// TwinCAT 3 PLC project Gesamtsystemebene
// ProgramVersion: 3.1.4024.0
// libraries:
//   Tc2_Standard, * (Beckhoff Automation GmbH)
//   Tc2_System, * (Beckhoff Automation GmbH)
//   Tc3_Module, * (Beckhoff Automation GmbH)
//   Tc3_PLCopen_OpcUa, * (Beckhoff Automation GmbH)
//   VisuDialogs, * (System)
//   Tc2_OpcUa,3.3.2.0,Beckhoff Automation GmbH
// project tree:
//   DUTs/01_Schnittstellen/ I_Auswertung.TcIO, I_Reaktor.TcIO
//   DUTs/02_Strukturen/ LeitungControlWord.TcDUT, RezeptControlWord.TcDUT, RezeptStatusWord.TcDUT (not stored), SekControlWord.TcDUT (not stored), SystemStatusWord.TcDUT
//   / GlobalTextList.TcGTLO, PlcTask.TcTTO, Visualisierungsmanager.TcVMO (not stored), VISU_TASK.TcTTO
//   GVLs/01_OPC_UA/ GVL_OPC_UA.TcGVL
//   GVLs/ GVL.TcGVL
//   POUs/01_Rezept/ Rezept_1.TcPOU
//   POUs/02_Funktionsblock/ FB_Auswertung.TcPOU, FB_Reaktoreinheit.TcPOU, FB_UpdateHandler.TcPOU
//   POUs/03_System/ Reaktoranlage.TcPOU, Systemauswertung.TcPOU
//   POUs/04_Abläufe/01_Vererbung/ FB_Basis.TcPOU
//   POUs/04_Abläufe/ FB_Lesen.TcPOU, FB_Trennen.TcPOU, FB_UpdateSek.TcPOU, FB_UpdateSys.TcPOU, FB_Verbinden.TcPOU, FB_Grundablauf.TcPOU
//   POUs/05_Kommunikation/ Connect.TcPOU, Disconnect.TcPOU, Read.TcPOU, UpdateSek.TcPOU, UpdateSys.TcPOU
//   POUs/ MAIN.TcPOU
//   VISUs/ Test_Visu.TcVIS
// real-time tasks:
//   TASK PlcTask: cycle T#10ms, priority 20, ADS port 350
//   TASK VISU_TASK: cycle T#200000us, priority 30, ADS port 351
//   TASK Gerät 1 (OPC UA Virtual)_Task_58: cycle T#40ms, priority 58, ADS port 352

CONFIGURATION Gesamtsystemebene
    RESOURCE PLC ON TwinCAT3
        TASK PlcTask(INTERVAL := T#10ms, PRIORITY := 20);
        TASK VISU_TASK(INTERVAL := T#200000us, PRIORITY := 30);
        PROGRAM MAIN WITH PlcTask : MAIN;
        PROGRAM VisuElems_Visu_Prg WITH VISU_TASK : VisuElems.Visu_Prg;
    END_RESOURCE
END_CONFIGURATION

// ---- DUTs/02_Strukturen/LeitungControlWord.TcDUT
TYPE LeitungControlWord :
STRUCT
	A_Prueft			:BOOL;
	A_Besetzt			:BOOL;
	B_Prueft			:BOOL;
	B_Besetzt			:BOOL;
	C_Prueft			:BOOL;
	C_Besetzt			:BOOL;
	D_Prueft			:BOOL;
	D_Besetzt			:BOOL;
	E_Prueft			:BOOL;
	E_Besetzt			:BOOL;
	F_Prueft			:BOOL;
	F_Besetzt			:BOOL;
END_STRUCT
END_TYPE

// ---- DUTs/02_Strukturen/RezeptControlWord.TcDUT
TYPE RezeptControlWord :
STRUCT			
	PowerOn			:BOOL;			// Einschalten von Reaktoreinheit
	SekReakt		:INT;			// Definierter sekundär-Reaktor
	Leitung			:INT;			// Definiert welche Leitung verwendet wird
	Temp			:REAL;			// Definierte Temperatur für Heiz- / Kühlprozess
	Enlteermenge	:REAL;			// Zu entleerende Menge
	Pumpmenge		:REAL;			// Zu pumpende Menge
	Haltedauer		:INT;			// Wie lange soll Temperatur gehalten werden (Faktor für Sekunden)
	Ruehrdauer		:INT;			// Wie lange soll gerührt werden (Faktor für Sekunden)
	Wartedauer		:INT;			// Wie lange soll gerührt werden (Faktor für Sekunden)
	Zirkulierdauer	:INT;			// Wie lange soll zirkuliert werden (Faktor für Sekunden)
END_STRUCT
END_TYPE

// ---- DUTs/02_Strukturen/SystemStatusWord.TcDUT
TYPE SystemStatusWord :
STRUCT
	// Das SystemStatusWord ist für die Interaktion zwischen den Reaktoren 	

	// Reaktor 1
	R1_Ready		:BOOL;
	R1_Activ		:BOOL;
	// Reaktor 2
	R2_Ready		:BOOL;
	R2_Activ		:BOOL;
	// Reaktor 3
	R3_Ready		:BOOL;
	R3_Activ		:BOOL;
	// Reaktor 4
	R4_Ready		:BOOL;
	R4_Activ		:BOOL;
	// Reaktor 5
	R5_Ready		:BOOL;
	R5_Activ		:BOOL;
	// Reaktor 6
	R6_Ready		:BOOL;
	R6_Activ		:BOOL;
	// Reaktor 7
	R7_Ready		:BOOL;
	R7_Activ		:BOOL;
END_STRUCT	
END_TYPE

// ---- GVLs/01_OPC_UA/GVL_OPC_UA.TcGVL
{attribute 'qualified_only'}
VAR_GLOBAL
	// Verbindungsinformationen
	IP 				:ARRAY [0..6] OF STRING := [
		        'opc.tcp://169.254.240.1:4840', 
        		'opc.tcp://169.254.240.2:4840',
				'opc.tcp://169.254.240.3:4840', 
				'opc.tcp://169.254.240.4:4840', 
				'opc.tcp://169.254.240.5:4840', 
 				'opc.tcp://169.254.240.6:4840', 
        		'opc.tcp://169.254.240.7:4840'];	
	NameSpace		:STRING(MAX_STRING_LENGTH) := 'urn:BeckhoffAutomation:Ua:PLC1';
	ConnectionHdl	:ARRAY [0..6] OF DWORD := [];
END_VAR

// ---- GVLs/GVL.TcGVL
{attribute 'qualified_only'}
VAR_GLOBAL
		
	// Rezeptparameter
	R1_CW			:RezeptControlWord;				// Lokale definierung der Parameter
	R1_SW			:RezeptStatusWord;				// Statusword für internen Handling
	
	R2_CW			:RezeptControlWord;				// Lokale definierung der Parameter
	R2_SW			:RezeptStatusWord;				// Statusword für internen Handling
	
	R3_CW			:RezeptControlWord;				// Lokale definierung der Parameter
	R3_SW			:RezeptStatusWord;				// Statusword für internen Handling
	
	R4_CW			:RezeptControlWord;				// Lokale definierung der Parameter
	R4_SW			:RezeptStatusWord;				// Statusword für internen Handling
	
	R5_CW			:RezeptControlWord;				// Lokale definierung der Parameter
	R5_SW			:RezeptStatusWord;				// Statusword für internen Handling
	
	R6_CW			:RezeptControlWord;				// Lokale definierung der Parameter
	R6_SW			:RezeptStatusWord;				// Statusword für internen Handling
	
	R7_CW			:RezeptControlWord;				// Lokale definierung der Parameter
	R7_SW			:RezeptStatusWord;				// Statusword für internen Handling
	
	
	// Leitungs-Control-Word
	
	// SekundärControlWord
	SekControlWord	:SekControlWord;

	// SystemStatusWord
	SysStatusWord	:SystemStatusWord;
	
	// Funktionsvariablen
	// 0 = System nicht verbunden
	// 1 = System teilweisen Verbunden (Nicht Aktiv)
	// 2 = System Aktiv (Prozess läuft)
	// 9 = Error
	SysState		:INT;						
	
	// Bedienparameter 
	Start			:BOOL;
	Connect			:BOOL;
	Disconnect		:BOOL;
	Read			:BOOL;
	
	SekUpdate_1		:BOOL;
	SekUpdate_2		:BOOL;
	SekUpdate_3		:BOOL;
	SekUpdate_4		:BOOL;
	SekUpdate_5		:BOOL;
	SekUpdate_6		:BOOL;
	SekUpdate_7		:BOOL;
	SysUpdate_1		:BOOL;
	SysUpdate_2		:BOOL;
	SysUpdate_3		:BOOL;
	SysUpdate_4		:BOOL;
	SysUpdate_5		:BOOL;
	SysUpdate_6		:BOOL;
	SysUpdate_7		:BOOL;
	SekUpdateReset	:BOOL;
	SysUpdateReset	:BOOL;
	
	
	// Zustands-Variablen
	Error			:BOOL;
	ErrorID			:DWORD;
	
END_VAR

// ---- DUTs/01_Schnittstellen/I_Auswertung.TcIO
INTERFACE I_Auswertung

METHOD M_STATUS_SEK : BOOL
VAR_INPUT
END_VAR
END_METHOD

METHOD M_STATUS_SYSTEM : BOOL
VAR_INPUT
END_VAR
END_METHOD

METHOD M_TRENNEN : BOOL
VAR_INPUT
END_VAR
END_METHOD

METHOD M_VERBINDEN : BOOL
VAR_INPUT
END_VAR
END_METHOD

PROPERTY P_Status : INT
GET
END_GET
END_PROPERTY

END_INTERFACE

// ---- DUTs/01_Schnittstellen/I_Reaktor.TcIO
INTERFACE I_Reaktor

METHOD M_LESEN : BOOL
VAR_INPUT
END_VAR
END_METHOD

METHOD M_SCHREIBEN : BOOL
VAR_INPUT
END_VAR
END_METHOD

METHOD M_TRENNEN : BOOL
VAR_INPUT
END_VAR
END_METHOD

METHOD M_VERBINDEN : BOOL
VAR_INPUT
END_VAR
END_METHOD

METHOD M_ZUSTAND : BOOL
VAR_INPUT
END_VAR
END_METHOD

PROPERTY P_Status : INT
GET
END_GET
END_PROPERTY

END_INTERFACE

// ---- POUs/MAIN.TcPOU
PROGRAM MAIN
VAR
END_VAR

VAR_INPUT
END_VAR

// Starten der Anlage
Reaktoranlage();
Systemauswertung();

// Starten des Kommunikationsauswertung
Connect();
Disconnect();

// Lesen von RezeptStatusWord
Read();

// Auswertung des RezeptControlWords für Sekundärreaktor
UpdateSek();

// Auswertung des RezeptStatusWords für Systemupdate
UpdateSys();

// Starten des Rezeptes
Rezept_1();

END_PROGRAM

// ---- POUs/03_System/Reaktoranlage.TcPOU
PROGRAM Reaktoranlage
VAR
	R1				:FB_Reaktoreinheit;
	R2				:FB_Reaktoreinheit;
	
	// Instanziierung von Switchfunktion für Update-Variable
	Switch_R1		:FB_UpdateHandler;
	Switch_R2		:FB_UpdateHandler;
	Switch_R3		:FB_UpdateHandler;
	Switch_R4		:FB_UpdateHandler;
	Switch_R5		:FB_UpdateHandler;
	Switch_R6		:FB_UpdateHandler;
	Switch_R7		:FB_UpdateHandler;
END_VAR

Switch_R1(
    I_SekUpdate := R1.O_SekUpdate,
    I_SekReset := GVL.SekUpdateReset,
    I_SysUpdate := R1.O_SysUpdate,
    I_SysReset := GVL.SysUpdateReset); // FB_UpdateHandler
GVL.ErrorID := R1.O_ErrorID;
GVL_OPC_UA.ConnectionHdl[0] := R1.O_ConnectionHdl;
GVL.SekUpdate_1 := Switch_R1.O_SekUpdate;
R2(I_RNr := 2, I_IP := GVL_OPC_UA.IP, I_NameSpace := GVL_OPC_UA.NameSpace, I_CW := GVL.R2_CW); // FB_Reaktoreinheit
GVL.Error := R2.O_Error;
GVL.ErrorID := R2.O_ErrorID;
GVL.R2_SW := R2.O_SW;
GVL_OPC_UA.ConnectionHdl[1] := R2.O_ConnectionHdl;
GVL.SekUpdate_2 := Switch_R2.O_SekUpdate;
Switch_R2(
    I_SekUpdate := R2.O_SekUpdate,
    I_SekReset := GVL.SekUpdateReset,
    I_SysUpdate := R2.O_SysUpdate,
    I_SysReset := GVL.SysUpdateReset); // FB_UpdateHandler
GVL.SysUpdate_1 := Switch_R1.O_SysUpdate;
GVL.SysUpdate_2 := Switch_R2.O_SysUpdate;
R1(I_RNr := 1, I_IP := GVL_OPC_UA.IP, I_NameSpace := GVL_OPC_UA.NameSpace, I_CW := GVL.R1_CW); // FB_Reaktoreinheit
GVL.Error := R1.O_Error;
GVL.R1_SW := R1.O_SW;

END_PROGRAM

// ---- POUs/02_Funktionsblock/FB_Reaktoreinheit.TcPOU
FUNCTION_BLOCK FB_Reaktoreinheit IMPLEMENTS I_Reaktor
VAR_INPUT
	I_RNr					:INT;						// Nummer für korrekte Zuweisung von SystemStatusWord
	I_IP					:ARRAY [0..6] OF STRING;
	I_NameSpace				:STRING(MAX_STRING_LENGTH);
	I_CW					:RezeptControlWord;			// Variable für Kommunikations-Schnittstelle (Write)					
END_VAR
	
VAR_OUTPUT
	O_Verbunden				:BOOL;
	O_SekUpdate				:BOOL;
	O_SysUpdate				:BOOL;
	O_ConnectionHdl			:DWORD;
	O_Error					:BOOL;
	O_ErrorID				:DWORD;
	O_SW					:RezeptStatusWord; 			// Statusword für Kontrolle des Rezeptes 
END_VAR

VAR
	V_Status				:INT;						// Interne Variable
	OPC_Status				:INT;						// Variable für Verbindugsprozess
	Counter					:INT := 0;
	
	// Instanziierung der Kommunikationsfunktionsblöcke
	Connect					:UA_Connect;
	NameSpaceInd			:UA_GetNamespaceIndex;
	Node					:UA_NodeGetHandle;
	NodeRelease				:UA_NodeReleaseHandle;
	Disconnect				:UA_Disconnect;
	Status					:UA_ConnectGetStatus;
	Read					:UA_Read;	
	Write					:UA_Write;
	
	// Instanziierung der relevanten Input-Variablen
	ConnectInfo				:ST_UASessionConnectInfo;			// Informationen für Verbindungsaufbau 
	NodeID_SW				:ST_UANodeID;
	NodeID_CW				:ST_UANodeID;
	NodeIdentifier_SW		:STRING(MAX_STRING_LENGTH) := 'GVL_OPC_UA.SW';
	NodeIdentifier_CW 		:ARRAY [0..9] OF STRING := [
        'GVL_OPC_UA.CW.PowerOn', 
        'GVL_OPC_UA.CW.SekReakt', 
        'GVL_OPC_UA.CW.Leitung', 
        'GVL_OPC_UA.CW.Temp', 
        'GVL_OPC_UA.CW.Enlteermenge', 
        'GVL_OPC_UA.CW.Pumpmenge', 
        'GVL_OPC_UA.CW.Haltedauer', 
        'GVL_OPC_UA.CW.Ruehrdauer', 
        'GVL_OPC_UA.CW.Wartedauer', 
        'GVL_OPC_UA.CW.Zirkulierdauer'];
	
	// Instanziierung der relevanten Output-Variablen
	NameSpaceIndex			:UINT;
	NodeHdl_SW				:DWORD;						// Nodehandler für Statusword
	NodeHdl_CW 				:ARRAY [0..9] OF DWORD := [];
	ConnectionStatus		:E_UAConnectionStatus;
	ServerState				:E_UAServerState;
	
	O_Sek: INT;
END_VAR

// Setzen der internen Variablen
V_Status := P_Status;

// OPC-UA-Schnittstelle:
CASE OPC_Status OF
0: // Idle
	O_SekUpdate := FALSE;
	O_SysUpdate := FALSE;
1:	// Connect
	// Definition der Verbindungsinformationen
	ConnectInfo.tSessionTimeout := T#1M;
	ConnectInfo.tConnectTimeout := T#1M;
	ConnectInfo.sApplicationName := '';
	ConnectInfo.eSecurityMode := eUASecurityMsgMode_Sign_Encrypt;				// 3 = Sign_Encrypted
	ConnectInfo.eSecurityPolicyUri := eUASecurityPolicy_Basic256Sha256;			// 4 = Basic256  
	ConnectInfo.eTransportProfileUri := eUATransportProfileUri_UATcp;			// 1 = UATcp
	ConnectInfo.stUserIdentTokenType.eUserIdentTokenType := eUAUITT_Username;	// 1 = Username
	ConnectInfo.stUserIdentTokenType.sTokenParam1 := 'Administrator';			// Username
	ConnectInfo.stUserIdentTokenType.sTokenParam2 := '1';						// PW

	// Verbinden zu OPC-UA-Schnittstelle
	Connect(Execute := TRUE, 
			ServerUrl := I_IP[I_RNr - 1], 
			SessionConnectInfo := ConnectInfo, 
			Timeout := T#5S, 
			ConnectionHdl => O_ConnectionHdl, 
			Error => O_Error, 
			ErrorID => O_ErrorID);
			
	IF NOT Connect.Busy THEN
		Connect(Execute := FALSE);
	END_IF
			
	IF Connect.Error THEN
		O_Verbunden := FALSE;
		OPC_Status := 0;
	END_IF
			
	IF Connect.Done THEN
		OPC_Status := 2;
	END_IF
			
//==================================================================================================
2:	// NameSpaceIndex
	NameSpaceInd(Execute := TRUE,
				ConnectionHdl := O_ConnectionHdl,
				NameSpaceUri := I_NameSpace,
				Timeout := T#5S,
				NameSpaceIndex => NameSpaceIndex, 
				Error => O_Error, 
				ErrorID => O_ErrorID);
				
	IF NOT NameSpaceInd.Busy THEN
		NameSpaceInd(Execute := FALSE);
	END_IF
				
	IF NameSpaceInd.Error THEN
		O_Verbunden := FALSE;
		OPC_Status := 0;
	END_IF
	
	IF NameSpaceInd.Done THEN
		OPC_Status := 3;
	END_IF

//==================================================================================================				
3: // Nodes
	// Definieren von relevanten Parameter
	// RezeptStatusword - SW
	NodeID_SW.eIdentifierType := eUAIdentifierType_String;
	NodeID_SW.nNamespaceIndex := NameSpaceIndex;
	NodeID_SW.sIdentifier := NodeIdentifier_SW;
	
	// Definieren von SW Node
	Node(Execute := TRUE,
			ConnectionHdl := O_ConnectionHdl,
			NodeID := NodeID_SW,
			Timeout := T#5S,
			NodeHdl => NodeHdl_SW, 
			Error => O_Error, 
			ErrorID => O_ErrorID);

	IF NOT Node.Busy THEN
		Node(Execute := FALSE);
	END_IF 		
	
	IF Node.Error THEN
		OPC_Status := 0;
	END_IF
	
	IF Node.Done THEN
		OPC_Status := 4;
	END_IF

//==================================================================================================		
4:	// RezeptControlword
	// Die Node-Identifier jeder Variable werden einzeln in ein Array geschrieben. 
	// Innerhalb des Cases gibt es  einen Counter der die Arrayposition managed
	// Dafür braucht es keine For-Schleife, da der instanziierte FB zyklisch ausgeführt wird
	
	NodeID_CW.eIdentifierType := eUAIdentifierType_String;
	NodeID_CW.nNamespaceIndex := NameSpaceIndex;
	NodeID_CW.sIdentifier := NodeIdentifier_CW[Counter];
	
	Node(Execute := TRUE,
			ConnectionHdl := O_ConnectionHdl,
			NodeID := NodeID_CW,
			Timeout := T#5S,
			NodeHdl => NodeHdl_CW[Counter], 
			Error => O_Error, 
			ErrorID => O_ErrorID);
			
	IF NOT Node.Busy THEN
		Node(Execute := FALSE);
	END_IF		
	
	IF Node.Error THEN
		OPC_Status := 0;
	END_IF
	
	IF Node.Done AND Counter < 9 THEN
		Counter := Counter + 1;
	END_IF
	
	IF Node.Done AND Counter > 8 THEN // Muss angepasst werden wegen case 5
		OPC_Status := 0; 
		Counter := 0;	
		O_Verbunden := TRUE;
	END_IF	

//==================================================================================================	
5: // Lesen von Variablen
	Read(Execute := TRUE,
		ConnectionHdl := O_ConnectionHdl,
		NodeHdl := NodeHdl_SW,
		pVariable := ADR(O_SW),
		cbData := SIZEOF(O_SW),
		Timeout := T#5S,
		Error => O_Error,
		ErrorID => O_ErrorID);
	
	IF NOT Read.Busy THEN
		Read(Execute := FALSE);
	END_IF	
		
	IF Read.Error THEN
		OPC_Status := 0;
	END_IF
	
	IF Read.Done THEN
		OPC_Status := 0;
		IF O_SW.ReactReady OR O_SW.ReactActiv THEN
			O_SysUpdate := TRUE;
		END_IF
	END_IF
	
//==================================================================================================	
6: // Schreiben von Variablen		
	// Jede Variable in der Struktur muss separat berschrieben werden. 
	// Ansonsten werden die Daten nicht korrekt übertragen.
	
	CASE Counter OF 
		0: 		Write.pVariable := ADR(I_CW.PowerOn);
				Write.cbData  := SIZEOF(I_CW.PowerOn);
		1: 		Write.pVariable := ADR(I_CW.SekReakt);
				Write.cbData  := SIZEOF(I_CW.SekReakt);
		2: 		Write.pVariable := ADR(I_CW.Leitung);
				Write.cbData  := SIZEOF(I_CW.Leitung);
		3: 		Write.pVariable := ADR(I_CW.Temp);
				Write.cbData  := SIZEOF(I_CW.Temp);
		4: 		Write.pVariable := ADR(I_CW.Enlteermenge);
				Write.cbData  := SIZEOF(I_CW.Enlteermenge);
		5: 		Write.pVariable := ADR(I_CW.Pumpmenge);
				Write.cbData  := SIZEOF(I_CW.Pumpmenge);
		6: 		Write.pVariable := ADR(I_CW.Haltedauer);
				Write.cbData  := SIZEOF(I_CW.Haltedauer);
		7: 		Write.pVariable := ADR(I_CW.Ruehrdauer);
				Write.cbData  := SIZEOF(I_CW.Ruehrdauer);
		8: 		Write.pVariable := ADR(I_CW.Wartedauer);
				Write.cbData  := SIZEOF(I_CW.Wartedauer);
		9: 		Write.pVariable := ADR(I_CW.Zirkulierdauer);
				Write.cbData  := SIZEOF(I_CW.Zirkulierdauer);
	END_CASE
	
	Write(Execute := TRUE,
		ConnectionHdl := O_ConnectionHdl,
		NodeHdl := NodeHdl_CW[Counter],
		Timeout := T#5S,
		Error => O_Error,
		ErrorID => O_ErrorID);
	
	IF NOT Write.Busy THEN
		Write(Execute := FALSE);
	END_IF	
		
	IF Write.Error THEN
		OPC_Status := 0;
	END_IF
	
	IF Write.Done AND Counter < 9 THEN
		Counter := Counter + 1;
	END_IF
	
	IF Write.Done AND Counter > 8 THEN
		Counter := 0;
		OPC_Status := 0;
		IF I_CW.SekReakt > 0 THEN
			O_SekUpdate := TRUE;
		END_IF
	END_IF

//==================================================================================================	
7: // Release Node - RezeptStatusword
	NodeRelease(Execute := TRUE,
				ConnectionHdl := O_ConnectionHdl,
				NodeHdl := NodeHdl_SW,
				Timeout := T#5S,
				Error => O_Error,
				ErrorID => O_ErrorID);
	
	IF NOT NodeRelease.Busy THEN
		NodeRelease(Execute := FALSE);
	END_IF
	
	IF NodeRelease.Error THEN
		OPC_Status := 0;
	END_IF

	IF NodeRelease.Done THEN
		OPC_Status := 8;
	END_IF			

//==================================================================================================
8:	// Release Node - RezeptControlword
	NodeRelease(Execute := TRUE,
				ConnectionHdl := O_ConnectionHdl,
				NodeHdl := NodeHdl_CW[Counter],
				Timeout := T#5S,
				Error => O_Error,
				ErrorID => O_ErrorID);
	
	IF NOT NodeRelease.Busy THEN
		NodeRelease(Execute := FALSE);
	END_IF	
	
	IF NodeRelease.Error THEN
		OPC_Status := 0;
	END_IF

	IF NodeRelease.Done AND Counter < 9 THEN
		Counter := Counter + 1;
	END_IF				
				
	IF NodeRelease.Done AND Counter > 8 THEN
		OPC_Status := 9;
	END_IF
	
//==================================================================================================
9: // Disconnect
	Disconnect(Execute := TRUE,
				ConnectionHdl := O_ConnectionHdl,
				Timeout := T#5S,
				Error => O_Error,
				ErrorID => O_ErrorID);
	
	IF NOT Disconnect.Busy THEN
		Disconnect(Execute := FALSE);
	END_IF	

	IF Disconnect.Error THEN
		OPC_Status := 0;
	END_IF		
				
	IF Disconnect.Done THEN
		O_Verbunden := FALSE;
		OPC_Status := 0;
	END_IF	

//==================================================================================================
10: // Verbingungsstatus
	Status(Execute := TRUE,
			ConnectionHdl := O_ConnectionHdl,
			GetServiceLevel := FALSE,
			Timeout := T#5S,
			Error => O_Error,
			ErrorID => O_ErrorID,
			ConnectionStatus => ConnectionStatus,
			ServerState => ServerState);
	
	IF Status.Error THEN
		OPC_Status := 0;
	END_IF		
		
	IF Status.Done THEN
		Status(Execute := FALSE);
		OPC_Status := 0;
	END_IF
	
END_CASE

METHOD M_LESEN : BOOL
VAR_INPUT
END_VAR
OPC_Status := 5;

IF Read.Done THEN
	M_LESEN := TRUE;
END_IF
END_METHOD

METHOD M_SCHREIBEN : BOOL
VAR_INPUT
END_VAR
OPC_Status := 6;

IF Write.Done THEN
	M_SCHREIBEN := TRUE;
END_IF
END_METHOD

METHOD M_TRENNEN : BOOL
VAR_INPUT
END_VAR
OPC_Status := 7;

IF Disconnect.Done THEN
	M_TRENNEN := TRUE;
END_IF
END_METHOD

METHOD M_VERBINDEN : BOOL
VAR_INPUT
END_VAR
OPC_Status := 1;

IF Node.Done THEN	
	M_VERBINDEN := TRUE;
END_IF
END_METHOD

METHOD M_ZUSTAND : BOOL
VAR_INPUT
END_VAR
OPC_Status := 10;

IF Status.Done THEN
	M_ZUSTAND := TRUE;
END_IF
END_METHOD

PROPERTY P_Status : INT
GET
// Status = 0: System nicht verbunden
// Status = 1: System verbunden
// Status = 2: System bereit für Kommunikation
// Status = 3: System eingeschalten
// Status = 4: Reaktor ready
// Status = 5: Reaktor läuft
// Status = 6: Statusword wurde gelesen
// Status = 9: Error

IF O_Verbunden THEN				
	P_Status := 1;
	
	IF O_SW.SysReady THEN
		P_Status := 2;
		
		IF O_SW.SysActiv THEN
			P_Status := 3;
			
			IF O_SW.ReactReady THEN
				P_Status := 4;
				
				IF O_SW.ReactActiv THEN
					P_Status := 5;
				END_IF
			END_IF
		END_IF
	END_IF
	IF Read.Done THEN
		P_Status := 6;
	END_IF
ELSE
	P_Status := 0;
END_IF

IF O_Error THEN
	P_Status := 9;
END_IF
END_GET
END_PROPERTY

END_FUNCTION_BLOCK

// ---- POUs/05_Kommunikation/Connect.TcPOU
PROGRAM Connect
VAR
	Connect_R1			:FB_Verbinden;
	Connect_R2			:FB_Verbinden;
	Connect_R3			:FB_Verbinden;
	Connect_R4			:FB_Verbinden;
	Connect_R5			:FB_Verbinden;
	Connect_R6			:FB_Verbinden;
	Connect_R7			:FB_Verbinden;
END_VAR

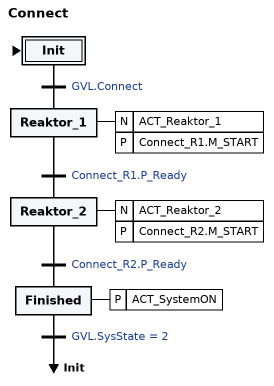
INITIAL_STEP Init:
END_STEP
TRANSITION FROM Init TO Reaktor_1
    := GVL.Connect;
END_TRANSITION
STEP Reaktor_1:
    ACT_Reaktor_1(N);
    Connect_R1.M_START(P);
END_STEP
TRANSITION FROM Reaktor_1 TO Reaktor_2
    := Connect_R1.P_Ready;
END_TRANSITION
STEP Reaktor_2:
    ACT_Reaktor_2(N);
    Connect_R2.M_START(P);
END_STEP
TRANSITION FROM Reaktor_2 TO Finished_
    := Connect_R2.P_Ready;
END_TRANSITION
STEP Finished_:  // name as stored: Finished 
    ACT_SystemON(P);
END_STEP
TRANSITION FROM Finished_ TO Init
    := GVL.SysState = 2;
END_TRANSITION

ACTION ACT_Reaktor_1:
Connect_R1(Reaktor := Reaktoranlage.R1, Auswertung := Systemauswertung.Auswertung_R1); // FB_Verbinden
END_ACTION

ACTION ACT_Reaktor_2:
Connect_R2(Reaktor := Reaktoranlage.R2, Auswertung := Systemauswertung.Auswertung_R2); // FB_Verbinden
END_ACTION

ACTION ACT_SystemON:
GVL.SysState := 2;
END_ACTION

END_PROGRAM

// ---- POUs/04_Abläufe/FB_Verbinden.TcPOU
FUNCTION_BLOCK FB_Verbinden EXTENDS FB_Basis
VAR_INPUT
	Reaktor			:I_Reaktor;
	Auswertung		:I_Auswertung;
END_VAR
VAR_OUTPUT
	
END_VAR
VAR
	
END_VAR

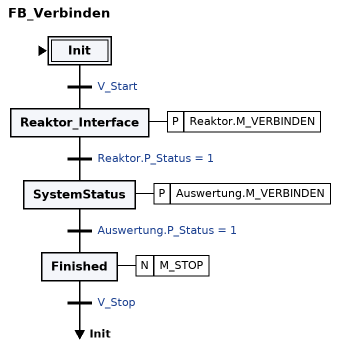
INITIAL_STEP Init:
END_STEP
TRANSITION FROM Init TO Reaktor_Interface
    := V_Start;
END_TRANSITION
STEP Reaktor_Interface:
    Reaktor.M_VERBINDEN(P);
END_STEP
TRANSITION FROM Reaktor_Interface TO SystemStatus_
    := Reaktor.P_Status = 1;
END_TRANSITION
STEP SystemStatus_:  // name as stored: SystemStatus 
    Auswertung.M_VERBINDEN(P);
END_STEP
TRANSITION FROM SystemStatus_ TO Finished
    := Auswertung.P_Status = 1;
END_TRANSITION
STEP Finished:
    M_STOP(N);
END_STEP
TRANSITION FROM Finished TO Init
    := V_Stop;
END_TRANSITION

END_FUNCTION_BLOCK

// ---- POUs/04_Abläufe/01_Vererbung/FB_Basis.TcPOU
FUNCTION_BLOCK FB_Basis
VAR_INPUT
END_VAR
VAR_OUTPUT
END_VAR
VAR
	V_Start			:BOOL;		// Variable für internes handling der Eigenschaft 
	V_Stop			:BOOL;		// Variable für internes handling der Eigenschaft 
END_VAR

METHOD M_START : BOOL
VAR_INPUT
END_VAR
V_Start := 1;
V_Stop := 0;
END_METHOD

METHOD M_STOP : BOOL
VAR_INPUT
END_VAR
V_Start := 0;
V_Stop := 1;
END_METHOD

PROPERTY P_Ready : BOOL
GET
P_Ready := V_Stop;
END_GET
END_PROPERTY

END_FUNCTION_BLOCK

// ---- POUs/03_System/Systemauswertung.TcPOU
PROGRAM Systemauswertung
VAR
	Auswertung_R1		:FB_Auswertung;
	Auswertung_R2		:FB_Auswertung;
END_VAR

GVL.Error := Auswertung_R1.O_Error;
GVL.ErrorID := Auswertung_R1.O_ErrorID;
GVL.SysStatusWord := Auswertung_R2.O_SysSW;
GVL.Error := Auswertung_R2.O_Error;
GVL.ErrorID := Auswertung_R2.O_ErrorID;
Auswertung_R1(
    I_RNr := 1,
    I_ConnectionHdl := GVL_OPC_UA.ConnectionHdl[0],
    I_NameSpace := GVL_OPC_UA.NameSpace,
    I_SW := GVL.R1_SW,
    I_SysSW := GVL.SysStatusWord,
    I_SekCW := GVL.SekControlWord); // FB_Auswertung
GVL.SysStatusWord := Auswertung_R1.O_SysSW;
Auswertung_R2(
    I_RNr := 2,
    I_ConnectionHdl := GVL_OPC_UA.ConnectionHdl[1],
    I_NameSpace := GVL_OPC_UA.NameSpace,
    I_SW := GVL.R2_SW,
    I_SysSW := GVL.SysStatusWord,
    I_SekCW := GVL.SekControlWord); // FB_Auswertung

END_PROGRAM

// ---- POUs/02_Funktionsblock/FB_Auswertung.TcPOU
FUNCTION_BLOCK FB_Auswertung IMPLEMENTS I_Auswertung
VAR_INPUT
	I_RNr				:INT;
	I_ConnectionHdl		:DWORD;
	I_NameSpace			:STRING(MAX_STRING_LENGTH);
	I_SW				:RezeptStatusWord;
	I_SysSW				:SystemStatusWord;
	I_SekCW				:SekControlWord;
END_VAR

VAR_OUTPUT
	O_Verbunden			:BOOL;
	O_SysSW				:SystemStatusWord;
	O_Error				:BOOL;
	O_ErrorID			:DWORD;
END_VAR

VAR
	V_Status				:INT;						// Interne Variable
	OPC_Status				:INT;
	SysSW					:SystemStatusWord;			// Variable für Handling von SystemStatusWord
	// Instanziierung der Kommunikationsfunktionsblöcke
	NameSpaceInd		:UA_GetNamespaceIndex;
	Node				:UA_NodeGetHandle;
	NodeRelease			:UA_NodeReleaseHandle;
	Write				:UA_Write;
	
	// Instanziierung der relevanten Input-Variablen
	NodeID_SysSW			:ST_UANodeID;
	NodeID_SekCW			:ST_UANodeID;
	NodeIdentifier_SysSW	:STRING(MAX_STRING_LENGTH) := 'GVL_OPC_UA.SysSW';
	NodeIdentifier_SekCW	:STRING(MAX_STRING_LENGTH) := 'GVL_OPC_UA.SekCW';
	
	// Instanziierung der relevanten Output-Variablen
	NameSpaceIndex			:UINT;
	NodeHdl_SysSW			:DWORD;	
	NodeHdl_SekCW			:DWORD;
	
END_VAR

// Setzen der internen Variablen
V_Status := P_Status;

CASE OPC_Status OF 
	0:	// Idle
	
	//==================================================================================================
	1: // GetNameSpace - SystemStatusWord
		NameSpaceInd(Execute := TRUE,
				ConnectionHdl := I_ConnectionHdl,
				NameSpaceUri := I_NameSpace,
				Timeout := T#5S,
				NameSpaceIndex => NameSpaceIndex, 
				Error => O_Error, 
				ErrorID => O_ErrorID);
					
		IF NOT NameSpaceInd.Busy THEN
			NameSpaceInd(Execute := FALSE);
		END_IF
					
		IF NameSpaceInd.Error THEN
			O_Verbunden := FALSE;
			OPC_Status := 0;
		END_IF
		
		IF NameSpaceInd.Done THEN
			OPC_Status := 2;
		END_IF
	
	//==================================================================================================
	2: // GetNode - SystemStatusWord
		NodeID_SysSW.eIdentifierType := eUAIdentifierType_String;
		NodeID_SysSW.nNamespaceIndex := NameSpaceIndex;
		NodeID_SysSW.sIdentifier := NodeIdentifier_SysSW;
	
		Node(Execute := TRUE,
				ConnectionHdl := I_ConnectionHdl,
				NodeID := NodeID_SysSW,
				Timeout := T#5S,
				NodeHdl => NodeHdl_SysSW, 
				Error => O_Error, 
				ErrorID => O_ErrorID);

		IF NOT Node.Busy THEN
			Node(Execute := FALSE);
		END_IF 		
		
		IF Node.Error THEN
			OPC_Status := 0;
		END_IF
		
		IF Node.Done THEN
			OPC_Status := 3; 	
		END_IF
		
	//==================================================================================================
	3: // GetNode - SekControlWord
		NodeID_SekCW.eIdentifierType := eUAIdentifierType_String;
		NodeID_SekCW.nNamespaceIndex := NameSpaceIndex;
		NodeID_SekCW.sIdentifier := NodeIdentifier_SekCW;
	
		// Definieren von SW Node
		Node(Execute := TRUE,
				ConnectionHdl := I_ConnectionHdl,
				NodeID := NodeID_SekCW,
				Timeout := T#5S,
				NodeHdl => NodeHdl_SekCW, 
				Error => O_Error, 
				ErrorID => O_ErrorID);

		IF NOT Node.Busy THEN
			Node(Execute := FALSE);
		END_IF 		
	
	IF Node.Error THEN
		OPC_Status := 0;
	END_IF
	
	IF Node.Done THEN
		OPC_Status := 0;
		O_Verbunden := TRUE;	
	END_IF
	
	//==================================================================================================
	4: // Beschreiben von SystemStatusWord auf allen Reaktoren
	   // Definieren des Zustandes des SystemSatusWords
	   
		CASE I_RNr OF 
			1:	SysSW.R1_Ready := I_SW.ReactReady;
				SysSW.R1_Activ := I_SW.ReactActiv;
				
			2:	SysSW.R2_Ready := I_SW.ReactReady;
				SysSW.R2_Activ := I_SW.ReactActiv;
				
			3:	SysSW.R3_Ready := I_SW.ReactReady;
				SysSW.R3_Activ := I_SW.ReactActiv;
				
			4:	SysSW.R4_Ready := I_SW.ReactReady;
				SysSW.R4_Activ := I_SW.ReactActiv;
				
			5:	SysSW.R5_Ready := I_SW.ReactReady;
				SysSW.R5_Activ := I_SW.ReactActiv;
				
			6:	SysSW.R6_Ready := I_SW.ReactReady;
				SysSW.R6_Activ := I_SW.ReactActiv;
				
			7:	SysSW.R7_Ready := I_SW.ReactReady;
				SysSW.R7_Activ := I_SW.ReactActiv;
		END_CASE
	
		// SystemStatusWord schreiben
		Write(Execute := TRUE,
			ConnectionHdl := I_ConnectionHdl,
			NodeHdl := NodeHdl_SysSW,
			pVariable := ADR(SysSW),
			cbData  := SIZEOF(SysSW),
			Timeout := T#5S,
			Error => O_Error,
			ErrorID => O_ErrorID);
			
		IF NOT Write.Busy THEN
			Write(Execute := FALSE);
		END_IF	
			
		IF Write.Error THEN
			OPC_Status := 0;
		END_IF
		
		IF Write.Done THEN
			O_SysSW := SysSW;
			OPC_Status := 0;
		END_IF	
	
	//==================================================================================================
	5: // Schreiben von Startvariablen für Sekundärreaktor
	
		// SystemStatusWord schreiben
		Write(Execute := TRUE,
			ConnectionHdl := I_ConnectionHdl,
			NodeHdl := NodeHdl_SekCW,
			pVariable := ADR(I_SekCW),
			cbData  := SIZEOF(I_SekCW),
			Timeout := T#5S,
			Error => O_Error,
			ErrorID => O_ErrorID);
		
		IF NOT Write.Busy THEN
			Write(Execute := FALSE);
		END_IF	
			
		IF Write.Error THEN
			OPC_Status := 0;
		END_IF
	
		IF Write.Done THEN
			OPC_Status := 0;
		END_IF	
		
	//==================================================================================================
	6: // ReleaseNode - SystemStatusWord
		NodeRelease(Execute := TRUE,
				ConnectionHdl := I_ConnectionHdl,
				NodeHdl := NodeHdl_SysSW,
				Timeout := T#5S,
				Error => O_Error,
				ErrorID => O_ErrorID);
	
		IF NOT NodeRelease.Busy THEN
			NodeRelease(Execute := FALSE);
		END_IF
		
		IF NodeRelease.Error THEN
			OPC_Status := 0;
		END_IF
	
		IF NodeRelease.Done THEN
			OPC_Status := 7;
		END_IF		
	//==================================================================================================
	7: // ReleaseNode - SekControlWord;
		NodeRelease(Execute := TRUE,
				ConnectionHdl := I_ConnectionHdl,
				NodeHdl := NodeHdl_SekCW,
				Timeout := T#5S,
				Error => O_Error,
				ErrorID => O_ErrorID);
	
		IF NOT NodeRelease.Busy THEN
			NodeRelease(Execute := FALSE);
		END_IF
		
		IF NodeRelease.Error THEN
			OPC_Status := 0;
		END_IF
	
		IF NodeRelease.Done THEN
			OPC_Status := 0;
		END_IF
END_CASE

METHOD M_STATUS_SEK : BOOL
VAR_INPUT
END_VAR
OPC_Status := 5;
END_METHOD

METHOD M_STATUS_SYSTEM : BOOL
VAR_INPUT
END_VAR
SysSW := I_SysSW;

OPC_Status := 4;
END_METHOD

METHOD M_TRENNEN : BOOL
VAR_INPUT
END_VAR
OPC_Status := 6;
END_METHOD

METHOD M_VERBINDEN : BOOL
VAR_INPUT
END_VAR
OPC_Status := 1;
END_METHOD

PROPERTY P_Status : INT
GET
// Status = 0: System nicht verbunden
// Status = 1: System verbunden
// Status = 2: System wurde beschrieben
// Status = 9: Error

IF O_Verbunden THEN
	P_Status := 1;
	
	IF Write.Done THEN
		P_Status := 2;
	END_IF
	
ELSE
	P_Status := 0;
END_IF

IF O_Error THEN
	P_Status := 9;
END_IF
END_GET
END_PROPERTY

END_FUNCTION_BLOCK

// ---- POUs/05_Kommunikation/Disconnect.TcPOU
PROGRAM Disconnect
VAR
	Disconnect_R1			:FB_Trennen;
	Disconnect_R2			:FB_Trennen;
	Disconnect_R3			:FB_Trennen;
	Disconnect_R4			:FB_Trennen;
	Disconnect_R5			:FB_Trennen;
	Disconnect_R6			:FB_Trennen;
	Disconnect_R7			:FB_Trennen;
END_VAR

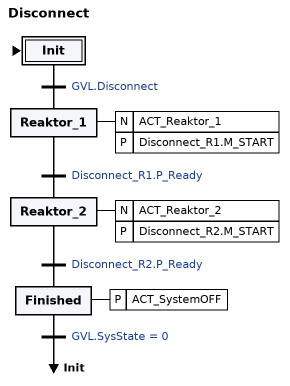
INITIAL_STEP Init:
END_STEP
TRANSITION FROM Init TO Reaktor_1
    := GVL.Disconnect;
END_TRANSITION
STEP Reaktor_1:
    ACT_Reaktor_1(N);
    Disconnect_R1.M_START(P);
END_STEP
TRANSITION FROM Reaktor_1 TO Reaktor_2
    := Disconnect_R1.P_Ready;
END_TRANSITION
STEP Reaktor_2:
    ACT_Reaktor_2(N);
    Disconnect_R2.M_START(P);
END_STEP
TRANSITION FROM Reaktor_2 TO Finished
    := Disconnect_R2.P_Ready;
END_TRANSITION
STEP Finished:
    ACT_SystemOFF(P);
END_STEP
TRANSITION FROM Finished TO Init
    := GVL.SysState = 0;
END_TRANSITION

ACTION ACT_Reaktor_1:
Disconnect_R1(Reaktor := Reaktoranlage.R1, Auswertung := Systemauswertung.Auswertung_R1); // FB_Trennen
END_ACTION

ACTION ACT_Reaktor_2:
Disconnect_R2(Reaktor := Reaktoranlage.R2, Auswertung := Systemauswertung.Auswertung_R2); // FB_Trennen
END_ACTION

ACTION ACT_SystemOFF:
GVL.SysState := 0;
END_ACTION

END_PROGRAM

// ---- POUs/04_Abläufe/FB_Trennen.TcPOU
FUNCTION_BLOCK FB_Trennen EXTENDS FB_Basis
VAR_INPUT
	Reaktor			:I_Reaktor;
	Auswertung		:I_Auswertung;
END_VAR
VAR_OUTPUT
END_VAR
VAR
	
END_VAR

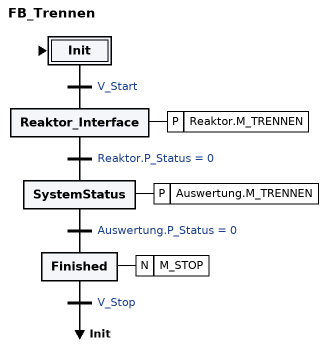
INITIAL_STEP Init:
END_STEP
TRANSITION FROM Init TO Reaktor_Interface
    := V_Start;
END_TRANSITION
STEP Reaktor_Interface:
    Reaktor.M_TRENNEN(P);
END_STEP
TRANSITION FROM Reaktor_Interface TO SystemStatus_
    := Reaktor.P_Status = 0;
END_TRANSITION
STEP SystemStatus_:  // name as stored: SystemStatus 
    Auswertung.M_TRENNEN(P);
END_STEP
TRANSITION FROM SystemStatus_ TO Finished
    := Auswertung.P_Status = 0;
END_TRANSITION
STEP Finished:
    M_STOP(N);
END_STEP
TRANSITION FROM Finished TO Init
    := V_Stop;
END_TRANSITION

END_FUNCTION_BLOCK

// ---- POUs/05_Kommunikation/Read.TcPOU
PROGRAM Read
VAR
	Read_R1				:FB_Lesen;
	Read_R2				:FB_Lesen;
	Read_R3				:FB_Lesen;
	Read_R4				:FB_Lesen;
	Read_R5				:FB_Lesen;
	Read_R6				:FB_Lesen;
	Read_R7				:FB_Lesen;
END_VAR

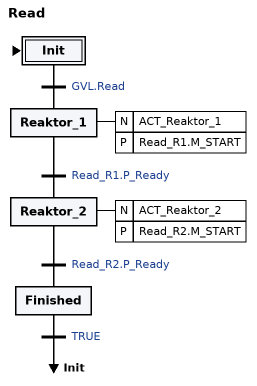
INITIAL_STEP Init:
END_STEP
TRANSITION FROM Init TO Reaktor_1
    := GVL.Read;
END_TRANSITION
STEP Reaktor_1:
    ACT_Reaktor_1(N);
    Read_R1.M_START(P);
END_STEP
TRANSITION FROM Reaktor_1 TO Reaktor_2
    := Read_R1.P_Ready;
END_TRANSITION
STEP Reaktor_2:
    ACT_Reaktor_2(N);
    Read_R2.M_START(P);
END_STEP
TRANSITION FROM Reaktor_2 TO Finished
    := Read_R2.P_Ready;
END_TRANSITION
STEP Finished:
END_STEP
TRANSITION FROM Finished TO Init
    := TRUE;
END_TRANSITION

ACTION ACT_Reaktor_1:
Read_R1(Reaktor := Reaktoranlage.R1); // FB_Lesen
END_ACTION

ACTION ACT_Reaktor_2:
Read_R2(Reaktor := Reaktoranlage.R2); // FB_Lesen
END_ACTION

END_PROGRAM

// ---- POUs/04_Abläufe/FB_Lesen.TcPOU
FUNCTION_BLOCK FB_Lesen EXTENDS FB_Basis
VAR_INPUT
	Reaktor			:I_Reaktor;
END_VAR

VAR_OUTPUT
END_VAR

VAR
END_VAR

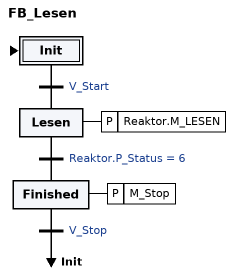
INITIAL_STEP Init:
END_STEP
TRANSITION FROM Init TO Lesen
    := V_Start;
END_TRANSITION
STEP Lesen:
    Reaktor.M_LESEN(P);
END_STEP
TRANSITION FROM Lesen TO Finished
    := Reaktor.P_Status = 6;
END_TRANSITION
STEP Finished:
    M_Stop(P);
END_STEP
TRANSITION FROM Finished TO Init
    := V_Stop;
END_TRANSITION

END_FUNCTION_BLOCK

// ---- POUs/02_Funktionsblock/FB_UpdateHandler.TcPOU
FUNCTION_BLOCK FB_UpdateHandler
VAR_INPUT
	I_SekUpdate			:BOOL;
	I_SekReset			:BOOL;
	I_SysUpdate			:BOOL;
	I_SysReset			:BOOL;
END_VAR

VAR_OUTPUT
	O_SekUpdate			:BOOL;
	O_SysUpdate			:BOOL;
END_VAR
VAR 
	SekSwitch			:SR;
	SysSwitch			:SR;
END_VAR

O_SekUpdate := SekSwitch.Q1;
SysSwitch(SET1 := I_SysUpdate, RESET := I_SysReset); // SR
O_SysUpdate := SysSwitch.Q1;
SekSwitch(SET1 := I_SekUpdate, RESET := I_SekReset); // SR

END_FUNCTION_BLOCK

// ---- POUs/05_Kommunikation/UpdateSek.TcPOU
PROGRAM UpdateSek
VAR
	SekUpdate_R1			:FB_UpdateSek;
	SekUpdate_R2			:FB_UpdateSek;
	SekUpdate_R3			:FB_UpdateSek;
	SekUpdate_R4			:FB_UpdateSek;
	SekUpdate_R5			:FB_UpdateSek;
	SekUpdate_R6			:FB_UpdateSek;
	SekUpdate_R7			:FB_UpdateSek;
END_VAR

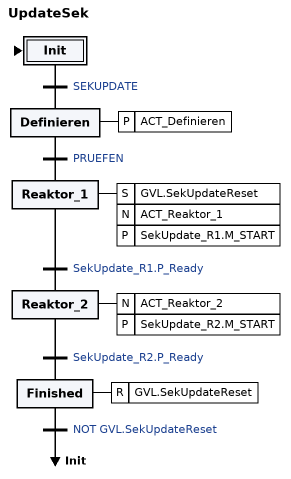
INITIAL_STEP Init:
END_STEP
TRANSITION FROM Init TO Definieren
    := SEKUPDATE;
END_TRANSITION
STEP Definieren:
    ACT_Definieren(P);
END_STEP
TRANSITION FROM Definieren TO Reaktor_1
    := PRUEFEN;
END_TRANSITION
STEP Reaktor_1:
    GVL.SekUpdateReset(S);
    ACT_Reaktor_1(N);
    SekUpdate_R1.M_START(P);
END_STEP
TRANSITION FROM Reaktor_1 TO Reaktor_2
    := SekUpdate_R1.P_Ready;
END_TRANSITION
STEP Reaktor_2:
    ACT_Reaktor_2(N);
    SekUpdate_R2.M_START(P);
END_STEP
TRANSITION FROM Reaktor_2 TO Finished
    := SekUpdate_R2.P_Ready;
END_TRANSITION
STEP Finished:
    GVL.SekUpdateReset(R);
END_STEP
TRANSITION FROM Finished TO Init
    := NOT GVL.SekUpdateReset;
END_TRANSITION

ACTION ACT_Definieren:
IF GVL.SekUpdate_1 THEN
	CASE GVL.R1_CW.SekReakt OF
		1:	GVL.SekControlWord.R1 := TRUE;
		2:	GVL.SekControlWord.R2 := TRUE;
		3:	GVL.SekControlWord.R3 := TRUE;
		4:	GVL.SekControlWord.R4 := TRUE;
		5:	GVL.SekControlWord.R5 := TRUE;
		6:	GVL.SekControlWord.R6 := TRUE;
		7:	GVL.SekControlWord.R7 := TRUE;
	END_CASE
END_IF

IF GVL.SekUpdate_2 THEN
	CASE GVL.R2_CW.SekReakt OF
		1:	GVL.SekControlWord.R1 := TRUE;
		2:	GVL.SekControlWord.R2 := TRUE;
		3:	GVL.SekControlWord.R3 := TRUE;
		4:	GVL.SekControlWord.R4 := TRUE;
		5:	GVL.SekControlWord.R5 := TRUE;
		6:	GVL.SekControlWord.R6 := TRUE;
		7:	GVL.SekControlWord.R7 := TRUE;
	END_CASE
END_IF

IF GVL.SekUpdate_3 THEN
	CASE GVL.R3_CW.SekReakt OF
		1:	GVL.SekControlWord.R1 := TRUE;
		2:	GVL.SekControlWord.R2 := TRUE;
		3:	GVL.SekControlWord.R3 := TRUE;
		4:	GVL.SekControlWord.R4 := TRUE;
		5:	GVL.SekControlWord.R5 := TRUE;
		6:	GVL.SekControlWord.R6 := TRUE;
		7:	GVL.SekControlWord.R7 := TRUE;
	END_CASE
END_IF

IF GVL.SekUpdate_4 THEN
	CASE GVL.R4_CW.SekReakt OF
		1:	GVL.SekControlWord.R1 := TRUE;
		2:	GVL.SekControlWord.R2 := TRUE;
		3:	GVL.SekControlWord.R3 := TRUE;
		4:	GVL.SekControlWord.R4 := TRUE;
		5:	GVL.SekControlWord.R5 := TRUE;
		6:	GVL.SekControlWord.R6 := TRUE;
		7:	GVL.SekControlWord.R7 := TRUE;
	END_CASE
END_IF

IF GVL.SekUpdate_5 THEN
	CASE GVL.R5_CW.SekReakt OF
		1:	GVL.SekControlWord.R1 := TRUE;
		2:	GVL.SekControlWord.R2 := TRUE;
		3:	GVL.SekControlWord.R3 := TRUE;
		4:	GVL.SekControlWord.R4 := TRUE;
		5:	GVL.SekControlWord.R5 := TRUE;
		6:	GVL.SekControlWord.R6 := TRUE;
		7:	GVL.SekControlWord.R7 := TRUE;
	END_CASE
END_IF

IF GVL.SekUpdate_6 THEN
	CASE GVL.R6_CW.SekReakt OF
		1:	GVL.SekControlWord.R1 := TRUE;
		2:	GVL.SekControlWord.R2 := TRUE;
		3:	GVL.SekControlWord.R3 := TRUE;
		4:	GVL.SekControlWord.R4 := TRUE;
		5:	GVL.SekControlWord.R5 := TRUE;
		6:	GVL.SekControlWord.R6 := TRUE;
		7:	GVL.SekControlWord.R7 := TRUE;
	END_CASE
END_IF

IF GVL.SekUpdate_7 THEN
	CASE GVL.R7_CW.SekReakt OF
		1:	GVL.SekControlWord.R1 := TRUE;
		2:	GVL.SekControlWord.R2 := TRUE;
		3:	GVL.SekControlWord.R3 := TRUE;
		4:	GVL.SekControlWord.R4 := TRUE;
		5:	GVL.SekControlWord.R5 := TRUE;
		6:	GVL.SekControlWord.R6 := TRUE;
		7:	GVL.SekControlWord.R7 := TRUE;
	END_CASE
END_IF
END_ACTION

ACTION ACT_Reaktor_1:
SekUpdate_R1(Auswertung := Systemauswertung.Auswertung_R1); // FB_UpdateSek
END_ACTION

ACTION ACT_Reaktor_2:
SekUpdate_R2(Auswertung := Systemauswertung.Auswertung_R2); // FB_UpdateSek
END_ACTION

TRANSITION PRUEFEN:
IF GVL.SekControlWord.R1 OR GVL.SekControlWord.R2 OR GVL.SekControlWord.R3 OR GVL.SekControlWord.R4 OR GVL.SekControlWord.R5 OR GVL.SekControlWord.R6 OR GVL.SekControlWord.R7 THEN
	PRUEFEN := TRUE;
ELSE 
	PRUEFEN := FALSE;
END_IF
END_TRANSITION

TRANSITION SEKUPDATE:
IF GVL.SekUpdate_1 OR
	GVL.SekUpdate_2 OR
	GVL.SekUpdate_3 OR
	GVL.SekUpdate_4 OR
	GVL.SekUpdate_5 OR
	GVL.SekUpdate_6 OR
	GVL.SekUpdate_7 THEN
	
	SEKUPDATE := TRUE;
ELSE 
	SEKUPDATE := FALSE;
END_IF
END_TRANSITION

END_PROGRAM

// ---- POUs/04_Abläufe/FB_UpdateSek.TcPOU
FUNCTION_BLOCK FB_UpdateSek EXTENDS FB_Basis
VAR_INPUT
	Auswertung		:I_Auswertung;
END_VAR

VAR_OUTPUT
END_VAR

VAR
END_VAR

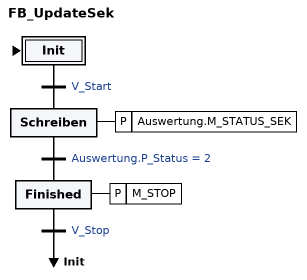
INITIAL_STEP Init:
END_STEP
TRANSITION FROM Init TO Schreiben
    := V_Start;
END_TRANSITION
STEP Schreiben:
    Auswertung.M_STATUS_SEK(P);
END_STEP
TRANSITION FROM Schreiben TO Finished
    := Auswertung.P_Status = 2;
END_TRANSITION
STEP Finished:
    M_STOP(P);
END_STEP
TRANSITION FROM Finished TO Init
    := V_Stop;
END_TRANSITION

END_FUNCTION_BLOCK

// ---- POUs/05_Kommunikation/UpdateSys.TcPOU
PROGRAM UpdateSys
VAR
	SysUpdate_R1			:FB_UpdateSys;
	SysUpdate_R2			:FB_UpdateSys;
	SysUpdate_R3			:FB_UpdateSys;
	SysUpdate_R4			:FB_UpdateSys;
	SysUpdate_R5			:FB_UpdateSys;
	SysUpdate_R6			:FB_UpdateSys;
	SysUpdate_R7			:FB_UpdateSys;
END_VAR

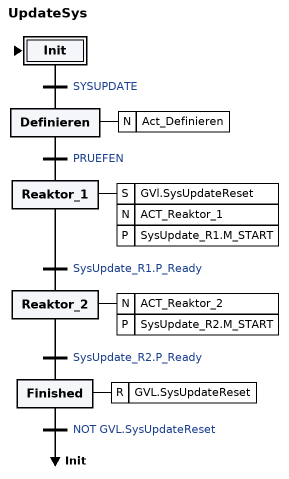
INITIAL_STEP Init:
END_STEP
TRANSITION FROM Init TO Definieren
    := SYSUPDATE;
END_TRANSITION
STEP Definieren:
    Act_Definieren(N);
END_STEP
TRANSITION FROM Definieren TO Reaktor_1
    := PRUEFEN;
END_TRANSITION
STEP Reaktor_1:
    GVl.SysUpdateReset(S);
    ACT_Reaktor_1(N);
    SysUpdate_R1.M_START(P);
END_STEP
TRANSITION FROM Reaktor_1 TO Reaktor_2
    := SysUpdate_R1.P_Ready;
END_TRANSITION
STEP Reaktor_2:
    ACT_Reaktor_2(N);
    SysUpdate_R2.M_START(P);
END_STEP
TRANSITION FROM Reaktor_2 TO Finished
    := SysUpdate_R2.P_Ready;
END_TRANSITION
STEP Finished:
    GVL.SysUpdateReset(R);
END_STEP
TRANSITION FROM Finished TO Init
    := NOT GVL.SysUpdateReset;
END_TRANSITION

ACTION ACT_Definieren:
IF GVL.SysUpdate_1 THEN
	IF GVL.R1_SW.ReactReady <> GVL.SysStatusWord.R1_Ready THEN
		GVL.SysStatusWord.R1_Ready := GVL.R1_SW.ReactReady;
	END_IF
	
	IF GVL.R1_SW.ReactActiv <> GVL.SysStatusWord.R1_Activ THEN
		GVL.SysStatusWord.R1_Activ := GVL.R1_SW.ReactActiv;
	END_IF
END_IF

IF GVL.SysUpdate_2 THEN
	IF GVL.R2_SW.ReactReady <> GVL.SysStatusWord.R2_Ready THEN
		GVL.SysStatusWord.R2_Ready := GVL.R2_SW.ReactReady;
	END_IF
	
	IF GVL.R2_SW.ReactActiv <> GVL.SysStatusWord.R2_Activ THEN
		GVL.SysStatusWord.R2_Activ := GVL.R2_SW.ReactActiv;
	END_IF
END_IF

IF GVL.SysUpdate_3 THEN
	IF GVL.R3_SW.ReactReady <> GVL.SysStatusWord.R3_Ready THEN
		GVL.SysStatusWord.R3_Ready := GVL.R3_SW.ReactReady;
	END_IF
	
	IF GVL.R3_SW.ReactActiv <> GVL.SysStatusWord.R3_Activ THEN
		GVL.SysStatusWord.R3_Activ := GVL.R3_SW.ReactActiv;
	END_IF
END_IF

IF GVL.SysUpdate_4 THEN
	IF GVL.R4_SW.ReactReady <> GVL.SysStatusWord.R4_Ready THEN
		GVL.SysStatusWord.R4_Ready := GVL.R4_SW.ReactReady;
	END_IF
	
	IF GVL.R4_SW.ReactActiv <> GVL.SysStatusWord.R4_Activ THEN
		GVL.SysStatusWord.R4_Activ := GVL.R4_SW.ReactActiv;
	END_IF
END_IF

IF GVL.SysUpdate_5 THEN
	IF GVL.R5_SW.ReactReady <> GVL.SysStatusWord.R5_Ready THEN
		GVL.SysStatusWord.R5_Ready := GVL.R5_SW.ReactReady;
	END_IF
	
	IF GVL.R5_SW.ReactActiv <> GVL.SysStatusWord.R5_Activ THEN
		GVL.SysStatusWord.R5_Activ := GVL.R5_SW.ReactActiv;
	END_IF
END_IF

IF GVL.SysUpdate_6 THEN
	IF GVL.R6_SW.ReactReady <> GVL.SysStatusWord.R6_Ready THEN
		GVL.SysStatusWord.R6_Ready := GVL.R6_SW.ReactReady;
	END_IF
	
	IF GVL.R6_SW.ReactActiv <> GVL.SysStatusWord.R6_Activ THEN
		GVL.SysStatusWord.R6_Activ := GVL.R6_SW.ReactActiv;
	END_IF
END_IF

IF GVL.SysUpdate_7 THEN
	IF GVL.R7_SW.ReactReady <> GVL.SysStatusWord.R7_Ready THEN
		GVL.SysStatusWord.R7_Ready := GVL.R7_SW.ReactReady;
	END_IF
	
	IF GVL.R7_SW.ReactActiv <> GVL.SysStatusWord.R7_Activ THEN
		GVL.SysStatusWord.R7_Activ := GVL.R7_SW.ReactActiv;
	END_IF
END_IF
END_ACTION

ACTION ACT_Reaktor_1:
SysUpdate_R1(Auswertung := Systemauswertung.Auswertung_R1); // FB_UpdateSys
END_ACTION

ACTION ACT_Reaktor_2:
SysUpdate_R2(Auswertung := Systemauswertung.Auswertung_R2); // FB_UpdateSys
END_ACTION

TRANSITION PRUEFEN:
IF GVL.SysUpdate_1 THEN
	IF GVL.R1_SW.ReactReady = GVL.SysStatusWord.R1_Ready AND GVL.R1_SW.ReactActiv = GVL.SysStatusWord.R1_Activ THEN
		PRUEFEN := TRUE;
	ELSE
		PRUEFEN := FALSE;
	END_IF
END_IF

IF GVL.SysUpdate_2 THEN
	IF GVL.R2_SW.ReactReady = GVL.SysStatusWord.R2_Ready AND GVL.R2_SW.ReactActiv = GVL.SysStatusWord.R2_Activ THEN
		PRUEFEN := TRUE;
	ELSE
		PRUEFEN := FALSE;
	END_IF
END_IF

IF GVL.SysUpdate_3 THEN
	IF GVL.R3_SW.ReactReady = GVL.SysStatusWord.R3_Ready AND GVL.R3_SW.ReactActiv = GVL.SysStatusWord.R3_Activ THEN
		PRUEFEN := TRUE;
	ELSE
		PRUEFEN := FALSE;
	END_IF
END_IF

IF GVL.SysUpdate_4 THEN
	IF GVL.R4_SW.ReactReady = GVL.SysStatusWord.R4_Ready AND GVL.R4_SW.ReactActiv = GVL.SysStatusWord.R4_Activ THEN
		PRUEFEN := TRUE;
	ELSE
		PRUEFEN := FALSE;
	END_IF
END_IF

IF GVL.SysUpdate_5 THEN
	IF GVL.R5_SW.ReactReady = GVL.SysStatusWord.R5_Ready AND GVL.R5_SW.ReactActiv = GVL.SysStatusWord.R5_Activ THEN
		PRUEFEN := TRUE;
	ELSE
		PRUEFEN := FALSE;
	END_IF
END_IF

IF GVL.SysUpdate_6 THEN
	IF GVL.R6_SW.ReactReady = GVL.SysStatusWord.R6_Ready AND GVL.R6_SW.ReactActiv = GVL.SysStatusWord.R6_Activ THEN
		PRUEFEN := TRUE;
	ELSE
		PRUEFEN := FALSE;
	END_IF
END_IF

IF GVL.SysUpdate_7 THEN
	IF GVL.R7_SW.ReactReady = GVL.SysStatusWord.R7_Ready AND GVL.R7_SW.ReactActiv = GVL.SysStatusWord.R7_Activ THEN
		PRUEFEN := TRUE;
	ELSE
		PRUEFEN := FALSE;
	END_IF
END_IF
END_TRANSITION

TRANSITION SYSUPDATE:
IF GVL.SysUpdate_1 OR
	GVL.SysUpdate_2 OR
	GVL.SysUpdate_3 OR
	GVL.SysUpdate_4 OR
	GVL.SysUpdate_5 OR
	GVL.SysUpdate_6 OR
	GVL.SysUpdate_7 THEN
	
	SYSUPDATE := TRUE;
ELSE 
	SYSUPDATE := FALSE;
END_IF
END_TRANSITION

END_PROGRAM

// ---- POUs/04_Abläufe/FB_UpdateSys.TcPOU
FUNCTION_BLOCK FB_UpdateSys EXTENDS FB_Basis
VAR_INPUT
	Auswertung		:I_Auswertung;
END_VAR

VAR_OUTPUT
END_VAR

VAR
END_VAR

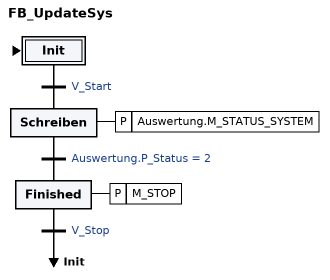
INITIAL_STEP Init:
END_STEP
TRANSITION FROM Init TO Schreiben
    := V_Start;
END_TRANSITION
STEP Schreiben:
    Auswertung.M_STATUS_SYSTEM(P);
END_STEP
TRANSITION FROM Schreiben TO Finished
    := Auswertung.P_Status = 2;
END_TRANSITION
STEP Finished:
    M_STOP(P);
END_STEP
TRANSITION FROM Finished TO Init
    := V_Stop;
END_TRANSITION

END_FUNCTION_BLOCK

// ---- POUs/01_Rezept/Rezept_1.TcPOU
PROGRAM Rezept_1
VAR
	// Abläufe
	GA_Reaktor_1		:FB_Grundablauf;
END_VAR

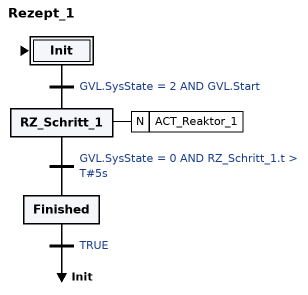
INITIAL_STEP Init:
END_STEP
TRANSITION FROM Init TO RZ_Schritt_1
    := GVL.SysState = 2 AND GVL.Start;
END_TRANSITION
STEP RZ_Schritt_1:
    ACT_Reaktor_1(N);
END_STEP
TRANSITION FROM RZ_Schritt_1 TO Finished
    := GVL.SysState = 0 AND RZ_Schritt_1.t > T#5s;
END_TRANSITION
STEP Finished:
END_STEP
TRANSITION FROM Finished TO Init
    := TRUE;
END_TRANSITION

ACTION ACT_Reaktor_1:
GA_Reaktor_1(Reaktor := Reaktoranlage.R1,
			SekReakt := 2,
			Temp := 0,
			Entleermenge := 50,
			Pumpmenge := 0,
			Haltedauer := 0,
			Ruehrdauer := 0,
			Wartedauer := 0,
			Zirkulierdauer := 0, 
			CW => GVL.R1_CW);
GA_Reaktor_1.M_START();
END_ACTION

END_PROGRAM

// ---- POUs/04_Abläufe/FB_Grundablauf.TcPOU
FUNCTION_BLOCK FB_Grundablauf EXTENDS FB_Basis
VAR_INPUT
	// Instanzieren von Reaktor mit Interface
	Reaktor			:I_Reaktor;
	
	// Prozessparameter
	SekReakt		:INT;
	Temp			:REAL;
	Entleermenge	:REAL;
	Pumpmenge		:REAL;
	Haltedauer		:INT;
	Ruehrdauer		:INT;
	Wartedauer		:INT;
	Zirkulierdauer	:INT;
END_VAR
VAR_OUTPUT
	CW				:RezeptControlWord;
END_VAR
VAR
	Leitung			:INT := 1;
	LeitungsCheck	:BOOL := TRUE;
END_VAR

